// TwinCAT 3 PLC project Plc
// Title: InvokeCSharp
// Company: Inxton
// Author: Inxton-Dev-Team
// ProjectVersion: 0.0.0.0
// ProgramVersion: 3.1.4023.0
// libraries:
//   Tc2_Standard, * (Beckhoff Automation GmbH)
//   Tc2_System, * (Beckhoff Automation GmbH)
//   Tc3_Module, * (Beckhoff Automation GmbH)
//   TcoCore, 0.5.0.829 (Vortex.Library)
//   TcoUtilities, 0.5.0.829 (Vortex.Library)
// project tree:
//   / PlcTask.TcTTO (not stored)
//   POUs/ App.TcPOU, MAIN.TcPOU (not stored)

// ---- POUs/App.TcPOU
FUNCTION_BLOCK App EXTENDS TcoCore.TcoContext
VAR
	i : INT;
END_VAR

(*~
	<docu>
		<summary>
			Main method of the TcoContext. This is the entry point of any control logic that belongs to this context. 
			The call of this method is ensured by calling the <c>InstanceName.Run()</c> method, and it must not be called explicitly.
			This method is abstract, and it must be overridden in derived block.
		</summary>
	</docu>
~*)
METHOD PROTECTED  Main
END_METHOD

END_FUNCTION_BLOCK
